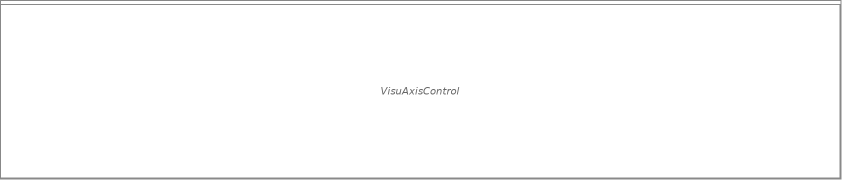
VISUALIZATION VisuAxisM3  // 842x180
    Frame (0,4 840x174)
        shows VisuAxisControl(sAxisName := sAxisM3_AName, stAxisVisu := stAxisM3_A)
END_VISUALIZATION

(* stored: Version 1.1.0.1, ProductVersion 3.1.4022.6
   Visu VisuAxisM3: Id {02255dba-7c3b-4e82-81bf-6b24afb60de4} *)
